(* CoDeSys 2.3.9.41 project: TRUBOGIB.pro *)
(* Libraries: STANDARD.LIB 4.10.05 11:14:46, IECSFC.LIB 13.4.06 15:51:28, ANALYZATION.LIB 5.10.99 09:05:06 *)

(* PLC configuration (modules and I/O channels)
PLC110_30 [Root] node -1, in %IB0 out %QB0 {ChannellName = PLC110-30_v2; MinCycleLength = 1; MaxCycleLength = 1000}
  Fast discrete inputs [I_SIMPLE_INPUT] node 0, in %IB0 out %QB0 {ChannellName = Fast discrete inputs; Filtrationtime = 10000}
    AT %IX0.0 [BitInput] Discrete input 1 {ChannellName = Enter name}
    AT %IX0.1 [BitInput] Discrete input 2 {ChannellName = Enter name}
  Discrete inputs - 16 [ID130] node 1, in %IB1 out %QB1 {ChannellName = Discrete inputs; Filtrationtime_GeneralINP = 10; PinCount = 16}
    AT %IB1.0 [ByteInput] 8 discrete inputs {ChannellName = Enter name}
    AT %IB1.1 [ByteInput] 8 discrete inputs {ChannellName = Enter name}
  Fast discrete outputs [OWEN_ID570] node 2, in %IB2 out %QB2 {ChannellName = Fast discrete outputs; SafeValueBool = FALSE; SafeValueBool = FALSE; SafeValueBool = FALSE; SafeValueBool = FALSE}
    AT %QX2.0 [BitOutput] Fast discrete output 1 {ChannellName = Enter name}
    AT %QX2.1 [BitOutput] Fast discrete output 2 {ChannellName = Enter name}
    AT %QX2.2 [BitOutput] Fast discrete output 3 {ChannellName = Enter name}
    AT %QX2.3 [BitOutput] Fast discrete output 4 {ChannellName = Enter name}
  Discrete outputs - 8 [ID131] node 3, in %IB3 out %QB3 {ChannellName = Discrete outputs; SafeValueByte = 0; Visibility = No; PinCount = 10}
    AT %QB3.0 [ByteOutput] 8 discrete outputs {ChannellName = Enter name}
  Special input [ID103] node 4, in %IB4 out %QB4 {ChannellName = Special input}
    AT %IX4.0 [BitInput] Special input {ChannellName = Enter name}
  Special output [ID104] node 5, in %IB5 out %QB5 {ChannellName = Special output}
    AT %QX5.0 [BitOutput] Special output {ChannellName = Enter name}
  ModBus (Master) [MODBUS_MASTER_ID450] node 6, in %IB6 out %QB6 {ChannellName = ModBus (Master); Visibility = No}
    AT %QD6.0 [DWordOutput] Last address {ChannellName = Enter name}
    AT %QW6.1 [WordOutput] Last error {ChannellName = Enter name}
    RS-485-1 [COM1_USART] node 0, in %IB6.0 out %QB6.0 {ChannellName = RS-485-1; CommunicationSpeed = 9600; Parity = NO PARITY CHECK; BitLength = 8 bits; StopLength = One stop bit; InterfaceType = RS485; FrameOriented = RTU; Timeout = 200; Visibility = No}
    Universal Modbus device [ID2000] node 1, in %IB6.1 out %QB6.1 {ChannellName = ESP8266; ModuleIP = 10:0:0:223; ServiceTimeout = 500; TCPport = 502; NetMode = Serial; ModuleSlaveAddress = 1; RequestType = By poll time; PeriodOfService = 100; Visibility = No; RepeatCounter = 0; ByteSequence = Trace_mode}
      AT %QB6.1.0 [ComChannel] Command (0xff - Start) {ChannellName = Enter name}
      Register output module [ID2004] node 0, in %IB6.1.0 out %QB6.1.0 {ChannellName = Register; ModbusAddress = 0; Command_write_one_reg = Write multiple registers(0x10); Visibility = No}
        mb_out_DefaultTarget AT %QW6.1.0.0 [WordOutput] {ChannellName = Enter name}
      Register output module [ID2004] node 1, in %IB6.1.1 out %QB6.1.1 {ChannellName = Register; ModbusAddress = 1; Command_write_one_reg = Write multiple registers(0x10); Visibility = No}
        mb_out_CurrentAngle AT %QW6.1.1.0 [WordOutput] {ChannellName = Enter name}
      Register output module [ID2004] node 2, in %IB6.1.2 out %QB6.1.2 {ChannellName = Register; ModbusAddress = 2; Command_write_one_reg = Write multiple registers(0x10); Visibility = No}
        mb_out_TargetAngle AT %QW6.1.2.0 [WordOutput] {ChannellName = Enter name}
      Register output module [ID2004] node 3, in %IB6.1.3 out %QB6.1.3 {ChannellName = Register; ModbusAddress = 3; Command_write_one_reg = Write multiple registers(0x10); Visibility = No}
        mb_out_Cycle AT %QW6.1.3.0 [WordOutput] {ChannellName = Enter name}
      Register output module [ID2004] node 4, in %IB6.1.4 out %QB6.1.4 {ChannellName = Register; ModbusAddress = 4; Command_write_one_reg = Write multiple registers(0x10); Visibility = No}
        mb_out_Done AT %QW6.1.4.0 [WordOutput] {ChannellName = Enter name}
      Register output module [ID2004] node 5, in %IB6.1.5 out %QB6.1.5 {ChannellName = Register; ModbusAddress = 5; Command_write_one_reg = Write multiple registers(0x10); Visibility = No}
        mb_out_Mode AT %QW6.1.5.0 [WordOutput] {ChannellName = Enter name}
      Register output module [ID2004] node 6, in %IB6.1.6 out %QB6.1.6 {ChannellName = Register; ModbusAddress = 6; Command_write_one_reg = Write multiple registers(0x10); Visibility = No}
        mb_out_Pedals AT %QW6.1.6.0 [WordOutput] {ChannellName = Enter name}
      Register input module [ID2003] node 7, in %IB6.1.7 out %QB6.1.7 {ChannellName = Register input module; ModbusAddress = 9; Command_read_regs = Read holding Registers  (0x03); Visibility = No}
        mb_in_Command AT %QW6.1.7.0 [WordOutput] {ChannellName = Enter name}
      Register input module [ID2003] node 8, in %IB6.1.8 out %QB6.1.8 {ChannellName = Register input module; ModbusAddress = 10; Command_read_regs = Read holding Registers  (0x03); Visibility = No}
        mb_in_WebTarget AT %QW6.1.8.0 [WordOutput] {ChannellName = Enter name}
*)

(* Global variable list: Global_Variables *)
VAR_GLOBAL RETAIN
    (* Inputs *)
    gDI_1   AT %IX0.0   : BOOL; (* Fast Input 1 *)
    gDI_2   AT %IX0.1   : BOOL; (* Fast Input 2 *)
    gDI_3   AT %IX1.0.0 : BOOL; (* Input 3 *)
    gDI_4   AT %IX1.0.1 : BOOL; (* Input 4 *)
    gDI_5   AT %IX1.0.2 : BOOL; (* Input 5 - Mode switch *)
    gDI_6   AT %IX1.0.3 : BOOL; (* Input 6 *)
    gDI_7   AT %IX1.0.4 : BOOL; (* Input 7 - Pedal Forward *)
    gDI_8   AT %IX1.0.5 : BOOL; (* Input 8 - Pedal Backward *)
    gDI_9   AT %IX1.0.6 : BOOL; (* Input 9 *)
    gDI_10  AT %IX1.0.7 : BOOL; (* Input 10 *)
    gDI_11  AT %IX1.1.0 : BOOL; (* Input 11 *)
    gDI_12  AT %IX1.1.1 : BOOL; (* Input 12 *)
    gDI_13  AT %IX1.1.2 : BOOL; (* Input 13 *)
    gDI_14  AT %IX1.1.3 : BOOL; (* Input 14 *)
    gDI_15  AT %IX1.1.4 : BOOL; (* Input 15 *)
    gDI_16  AT %IX1.1.5 : BOOL; (* Input 16 *)
    gDI_17  AT %IX1.1.6 : BOOL; (* Input 17 *)
    gDI_18  AT %IX1.1.7 : BOOL; (* Input 18 *)

    (* Encoder inputs *)
    gEncoderA AT %IX0.0 : BOOL;  (* Encoder A *)
    gEncoderB AT %IX0.1 : BOOL;  (* Encoder B *)

    (* Outputs *)
    gDO_1   AT %QX2.0   : BOOL; (* Fast Output 1 *)
    gDO_2   AT %QX2.1   : BOOL; (* Fast Output 2 *)
    gDO_3   AT %QX2.2   : BOOL; (* Fast Output 3 *)
    gDO_4   AT %QX2.3   : BOOL; (* Fast Output 4 *)
    gDO_5   AT %QX3.0.0 : BOOL; (* Output 5 *)
    gDO_6   AT %QX3.0.1 : BOOL; (* Output 6 *)
    gDO_7   AT %QX3.0.2 : BOOL; (* Output 7 *)
    gDO_8   AT %QX3.0.3 : BOOL; (* Output 8 *)
    gDO_9   AT %QX3.0.4 : BOOL; (* Output 9 *)
    gDO_10  AT %QX3.0.5 : BOOL; (* Output 10 - Motor Forward *)
    gDO_11  AT %QX3.0.6 : BOOL; (* Output 11 - Motor Backward *)
    gDO_12  AT %QX3.0.7 : BOOL; (* Output 12 - Target Pulse *)

    (* Beeper *)
    gBeeper AT %QX5.0   : BOOL; (* Beeper output *)

    (* ModBus Master *)
    gModbus_Master_Channel AT %QD6.0 : DWORD; (* Last address *)
    gModbus_Master_LastError AT %QW6.1 : WORD; (* Last error *)

    (* Internal state *)
    gTargetAngle : INT := 45;
    gDefaultTarget : INT := 45;
    gCurrentAngle : INT := 0;
    gCycle : INT := 1;
    gEncoderCount : DINT := 0;
    gCalibCountsPerRev : DINT := 360;
END_VAR

(* Data type *)
TYPE COMSETTINGS_FALLBACK : STRUCT
    Port : INT; (* PORTS in library; INT used locally to avoid enum conflicts *)
    dwBaudRate : DWORD;
    byStopBits : BYTE;
    byParity : BYTE;
    dwTimeout : DWORD;
    dwBufferSize : DWORD;
    dwScan : DWORD;
END_STRUCT
END_TYPE

(* POU PLC_PRG, ST *)
PROGRAM PLC_PRG
VAR
    (* First scan flag *)
    init_done : BOOL := FALSE;

    (* Control Inputs *)
    prev_d5 : BOOL;
    enableStart : BOOL;      (* D5: 1=Manual, 0=Auto *)
    btnD7 : BOOL;            (* D7: Pedal Forward *)
    btnD8 : BOOL;            (* D8: Pedal Backward *)
    both : BOOL;             (* Both pedals *)
    
    (* Encoder *)
    encAEdge : R_TRIG;
    encBEdge : R_TRIG;
    
    (* Process State *)
    done : BOOL := FALSE;    (* Target reached flag *)
    
    (* Timers & Triggers *)
    targetPulseTrigger : BOOL := FALSE;
    tpTarget : TP;           (* Pulse on DO12 *)
    beepTargetTrigger : BOOL := FALSE;
    tpBeepTarget : TP;       (* Beep on target reached *)
    
    errorBeepTrigger : BOOL := FALSE;
    tErrTotal : TON;
    tErrDelay1 : TON;
    tErrDelay2 : TON;
    tErrDelay3 : TON;
    rTrigErr1 : R_TRIG;
    rTrigErr2 : R_TRIG;
    rTrigErr3 : R_TRIG;
    tpErr : TP;

    (* Done auto-reset timer: holds done=TRUE for 500ms then resets *)
    tonDoneHold : TON;
    doneHolding : BOOL := FALSE;

    (* Change beep - 2 short beeps for: default angle change, mode switch *)
    changeBeepTrigger : BOOL := FALSE;
    tChangeTotal : TON;
    tChangeDelay1 : TON;
    tChangeDelay2 : TON;
    rTrigChange1 : R_TRIG;
    rTrigChange2 : R_TRIG;
    tpChangeBeep : TP;

    (* Edge detection for error beeps *)
    prev_d7 : BOOL := FALSE;
    prev_d8 : BOOL := FALSE;
    prev_both : BOOL := FALSE;

    (* Modbus command edge detection *)
    prev_mb_in_command : WORD := 0;
    prev_mb_in_WebTarget : WORD := 0;
END_VAR
(* 1. Input Mapping *)
enableStart := gDI_5; 
btnD7 := gDI_7;       
btnD8 := gDI_8;       
both := btnD7 AND btnD8;

(* 1.1 First scan init - prevent false edge detection *)
IF NOT init_done THEN
    prev_d5 := enableStart;
    prev_mb_in_WebTarget := mb_in_WebTarget;
    prev_mb_in_command := mb_in_Command;
    init_done := TRUE;
END_IF;

(* 2. Encoder Processing *)
encAEdge(CLK := gEncoderA);
encBEdge(CLK := gEncoderB);

IF encAEdge.Q THEN
    IF gEncoderB THEN
        gEncoderCount := gEncoderCount + 1;
    ELSE
        gEncoderCount := gEncoderCount - 1;
    END_IF;
END_IF;

(* 3. Angle Calculation - 360P/R encoder: 1 count = 1 degree *)
IF gCalibCountsPerRev = 0 THEN
    gCalibCountsPerRev := 360;
END_IF;
gCurrentAngle := DINT_TO_INT(gEncoderCount * 360 / gCalibCountsPerRev);

(* 4. Mode Switching - beep only, zero reset moved to web button *)
IF prev_d5 <> enableStart THEN
    changeBeepTrigger := TRUE;
    IF prev_d5 AND NOT enableStart THEN
        (* Manual->Auto: just prepare for auto mode, no zero reset *)
        gCycle := 1;
        gTargetAngle := gDefaultTarget;
        done := FALSE;
    END_IF;
END_IF;
prev_d5 := enableStart;

(* 5. Modbus / Web Commands Processing *)

(* 5.1 Web Target Update - register 10 - edge detection *)
(* ESP holds value for 500ms, then clears to 0 *)
(* PLC detects non-zero value different from prev *)
IF mb_in_WebTarget <> 0 AND mb_in_WebTarget <> prev_mb_in_WebTarget THEN
    gDefaultTarget := WORD_TO_INT(mb_in_WebTarget);
    gTargetAngle := gDefaultTarget;
    done := FALSE;
    gCycle := 1;
    changeBeepTrigger := TRUE;
END_IF;
prev_mb_in_WebTarget := mb_in_WebTarget;

(* 5.2 Command Register - register 9 *)
IF mb_in_Command <> 0 AND mb_in_Command <> prev_mb_in_command THEN
    CASE WORD_TO_INT(mb_in_Command) OF
        1: (* START *)
            IF NOT enableStart THEN done := FALSE; gCycle := 1; gTargetAngle := gDefaultTarget; END_IF;
        2: (* STOP *)
            done := TRUE;
        3: (* ZERO - full reset: zero encoder, set cycle 1, reset done *)
            gEncoderCount := 0;
            gCurrentAngle := 0;
            gCycle := 1;
            gTargetAngle := gDefaultTarget;
            done := FALSE;
            changeBeepTrigger := TRUE;
    END_CASE;
END_IF;
prev_mb_in_command := mb_in_Command;

(* 6. Cycle Logic (Auto Mode) *)
IF NOT enableStart AND NOT done THEN
    IF gCycle = 1 THEN
        gTargetAngle := gDefaultTarget;
    ELSIF gCycle = 2 THEN
        gTargetAngle := 0;
    END_IF;
END_IF;

(* 7. Output to Modbus (PLC -> ESP registers 0-6) *)
mb_out_DefaultTarget := INT_TO_WORD(gDefaultTarget);
mb_out_CurrentAngle  := INT_TO_WORD(gCurrentAngle);
mb_out_TargetAngle   := INT_TO_WORD(gTargetAngle);
mb_out_Cycle         := INT_TO_WORD(gCycle);

IF done THEN mb_out_Done := 1; ELSE mb_out_Done := 0; END_IF;
IF enableStart THEN mb_out_Mode := 1; ELSE mb_out_Mode := 0; END_IF;

mb_out_Pedals := 0;
IF btnD7 THEN mb_out_Pedals := mb_out_Pedals + 1; END_IF;
IF btnD8 THEN mb_out_Pedals := mb_out_Pedals + 2; END_IF;

(* 8. Motor Control Logic *)
IF enableStart THEN  (* MANUAL MODE *)
    gDO_10 := btnD7 AND NOT btnD8 AND NOT both;
    gDO_11 := btnD8 AND NOT btnD7 AND NOT both;
ELSE  (* AUTO MODE *)
    (* Cycle 1: bending - only forward allowed, backward jams tube *)
    (* Cycle 2: return  - only backward allowed, forward jams tube *)
    gDO_10 := btnD7 AND NOT btnD8 AND (gCurrentAngle < gTargetAngle) AND NOT done AND (gCycle = 1);
    gDO_11 := btnD8 AND NOT btnD7 AND (gCurrentAngle > 0) AND NOT done AND (gCycle = 2);
END_IF;

(* 9. Target Reached Check - directional, can't be missed by fast encoder *)
IF NOT enableStart AND NOT done THEN
    IF (gCycle = 1 AND gCurrentAngle >= gTargetAngle AND gTargetAngle > 0) THEN
        (* Cycle 1: forward bending reached or passed target *)
        done := TRUE;
        doneHolding := TRUE;
        targetPulseTrigger := TRUE;
        beepTargetTrigger := TRUE;
        gCycle := 2;
        gTargetAngle := 0;        (* Next target: return to zero *)
    ELSIF (gCycle = 2 AND gCurrentAngle <= gTargetAngle) THEN
        (* Cycle 2: backward return reached or passed zero *)
        done := TRUE;
        doneHolding := TRUE;
        targetPulseTrigger := TRUE;
        beepTargetTrigger := TRUE;
        gCycle := 1;
        gTargetAngle := gDefaultTarget; (* Next target: bend again *)
    END_IF;
END_IF;

(* 9.1 Done Auto-Reset: hold done=TRUE for 500ms pause, then allow next cycle *)
(* This gives operator time to release pedal and hear beep before next action *)
tonDoneHold(IN := doneHolding, PT := T#500MS);
IF tonDoneHold.Q THEN
    done := FALSE;
    doneHolding := FALSE;
END_IF;

(* 10. Indication & Beeper *)

(* Target Reached Pulse *)
tpTarget(IN := targetPulseTrigger, PT := T#500MS);
IF tpTarget.Q THEN targetPulseTrigger := FALSE; END_IF;

(* Success Beep - target reached (1 x 500ms) *)
(* Success Beep - target reached (1 x 200ms) *)
tpBeepTarget(IN := beepTargetTrigger, PT := T#200MS);

(* Error Conditions - auto mode, any cycle *)
IF NOT enableStart THEN
    (* Both pedals pressed *)
    IF both AND NOT prev_both THEN
        errorBeepTrigger := TRUE;
    END_IF;
    (* Forward pedal beyond limit or wrong cycle *)
    IF btnD7 AND NOT prev_d7 THEN
        IF gCurrentAngle >= gDefaultTarget OR gCycle = 2 THEN
            errorBeepTrigger := TRUE;
        END_IF;
    END_IF;
    (* Backward pedal at zero or wrong cycle *)
    IF btnD8 AND NOT prev_d8 THEN
        IF gCurrentAngle <= 0 OR gCycle = 1 THEN
            errorBeepTrigger := TRUE;
        END_IF;
    END_IF;
END_IF;

(* Error Beep Sequence (3 short beeps x 200ms) *)
tErrTotal(IN := errorBeepTrigger, PT := T#1400MS);
tErrDelay1(IN := errorBeepTrigger, PT := T#0MS);
tErrDelay2(IN := errorBeepTrigger, PT := T#400MS);
tErrDelay3(IN := errorBeepTrigger, PT := T#800MS);

rTrigErr1(CLK := tErrDelay1.Q);
rTrigErr2(CLK := tErrDelay2.Q);
rTrigErr3(CLK := tErrDelay3.Q);

tpErr(IN := (rTrigErr1.Q OR rTrigErr2.Q OR rTrigErr3.Q), PT := T#200MS);

(* Change Beep - default angle change / mode switch (2 x 150ms) *)
tChangeTotal(IN := changeBeepTrigger, PT := T#800MS);
tChangeDelay1(IN := changeBeepTrigger, PT := T#0MS);
tChangeDelay2(IN := changeBeepTrigger, PT := T#400MS);

rTrigChange1(CLK := tChangeDelay1.Q);
rTrigChange2(CLK := tChangeDelay2.Q);

tpChangeBeep(IN := (rTrigChange1.Q OR rTrigChange2.Q), PT := T#150MS);

(* Combined beeper output - ALL signals *)
gBeeper := tpBeepTarget.Q OR tpErr.Q OR tpChangeBeep.Q;

(* DO12 mirrors ALL beeper signals (external loud speaker) *)
gDO_12 := gBeeper;

IF tErrTotal.Q THEN errorBeepTrigger := FALSE; END_IF;
IF tChangeTotal.Q THEN changeBeepTrigger := FALSE; END_IF;
IF NOT tpBeepTarget.Q THEN beepTargetTrigger := FALSE; END_IF;

(* Update Previous States *)
prev_d7 := btnD7;
prev_d8 := btnD8;
prev_both := both;
END_PROGRAM
